INTERFACE I_Power  EXTENDS I_Output

METHOD Enables
VAR_INPUT
    Enable	: BOOL;
    Enable_Positive	: BOOL;
    Enable_Negative	: BOOL;
END_VAR
END_METHOD

PROPERTY Override : LREAL
GET
END_GET
END_PROPERTY

METHOD Power
VAR_INPUT
    Enable	: BOOL;
    Enable_Positive	: BOOL;
    Enable_Negative	: BOOL;
    Override	: LREAL := 100.0;
    BufferMode	: MC_BufferMode := MC_BufferMode.MC_Aborting;
END_VAR
END_METHOD

PROPERTY PowerIsEnabled : BOOL
GET
END_GET
END_PROPERTY

END_INTERFACE

(* stored: Version 1.1.0.1
   Itf I_Power: Id {3e27e6e8-6685-424d-9ead-eda513d1c175}
   Method Enables: Id {b68894a9-114b-4772-b0bc-887ad3b3442e}
   Property Override: Id {961843bf-f471-4df9-93bb-5367e5ad1298}
   Get Get: Id {680fd513-de2f-4508-bf7e-cee66bf848d5}
   Method Power: Id {6ec5953f-7853-4ae8-b7bf-ca6c5f20defd}
   Property PowerIsEnabled: Id {51943bc5-fd82-4d37-a623-d1f89afd6f2e}
   Get Get: Id {f6f920c1-2a15-45fb-99e2-22914eacf6cf} *)
